// TIA Portal V19 export
DATA_BLOCK "A0302_Spintore_PERS"   // DB76
// stored: MemoryReserve 100
   VAR RETAIN
      Par : Struct
         Sens : "Analogic_SensorManagement_Par";
      END_STRUCT;
      Data : Struct
         Sens : "Analogic_SensorManagement_Data";
         HMI { ExternalAccessible := 'False'; ExternalVisible := 'False'; ExternalWritable := 'False'} : "HMI_Preset";
         Ax_Pos : "A0301_Mach_Ax_Pos_Data";
      END_STRUCT;
      Par_Mach { S7_SetPoint := 'True'} : "A0301_Mach_Sens_Par";
      Par_Ax_Manu : "Positioning_EPOS_Machine_Par";
      Pers_Data : Struct
         EncoderAbsolute_Preset_OK : Bool := TRUE;
         Persistent_ActualPosition : LReal := 670.75;
      END_STRUCT;
      Par_Ax_Auto : "A0301_Mach_Speed_Par";
   END_VAR
BEGIN
   Par.Sens.Enable := TRUE;
   Par.Sens.RangeLow := 0.0;
   Par.Sens.RangeHigh := 150.0;
   Data.Sens.OffsetValue := 18.9832916259766;
   Data.Sens.OffsetValid := TRUE;
   Data.HMI.Button := FALSE;
   Data.HMI.Value := 150.0;
   Data.HMI.Feedback := 150.037933349609;
   Data.Ax_Pos.OffsetPosAttesa := 500.0;
   Data.Ax_Pos.PosAttesa := 670.75;
   Data.Ax_Pos.PosFineSpinta := 1170.75;
   Par_Mach.Tol_Work := 100.0;
   Par_Mach.WorkTime_SensDisable := T#100MS;
   Par_Ax_Manu.PosTolerance := 0.5;
   Par_Ax_Manu.DelayInPosition := T#10MS;
   Par_Ax_Manu.Man_Vel := 20000.0;
   Par_Ax_Manu.Man_Acc := 3000.0;
   Par_Ax_Manu.Man_Dec := 1000.0;
   Par_Ax_Auto.SemiAut_Vel := 25000.0;
   Par_Ax_Auto.Aut_Vel := 20000.0;
   Par_Ax_Auto.Aut_Acc := 3000.0;
   Par_Ax_Auto.Aut_Dec := 1000.0;
END_DATA_BLOCK
